// TIA Portal V19 export
VAR_GLOBAL   // PLC tag table "Tag table from XML_1"
   "At 1" AT %I0.0 : Bool;
   "At 2" AT %I0.1 : Bool;
   "At 3" AT %I0.2 : Bool;
   "At elevator" AT %I0.3 : Bool;
   "At entry" AT %I0.4 : Bool;
   "At exit" AT %I0.5 : Bool;
   "At 0 (low)" AT %I0.6 : Bool;
   "At 0 (high)" AT %I0.7 : Bool;
   "At 1 (low)" AT %I1.0 : Bool;
   "At 1 (high)" AT %I1.1 : Bool;
   "At 2 (low)" AT %I1.2 : Bool;
   "At 2 (high)" AT %I1.3 : Bool;
   "At 3 (low)" AT %I1.4 : Bool;
   "At 3 (high)" AT %I1.5 : Bool;
   Start AT %I1.6 : Bool;
   Reset AT %I1.7 : Bool;
   Stop AT %I2.0 : Bool;
   "Emergency stop" AT %I2.1 : Bool;
   Auto AT %I2.2 : Bool;
   "Diffuse Sensor 0" AT %I2.3 : Bool;
   "Diffuse Sensor 1" AT %I2.4 : Bool;
   "Diffuse Sensor 2" AT %I2.5 : Bool;
   "Diffuse Sensor 3" AT %I2.6 : Bool;
   "Conveyor 0" AT %Q0.0 : Bool;
   "Conveyor 1" AT %Q0.1 : Bool;
   "Conveyor 2" AT %Q0.2 : Bool;
   "Conveyor 3" AT %Q0.3 : Bool;
   "Exit conveyor" AT %Q0.4 : Bool;
   Load AT %Q0.5 : Bool;
   Unload AT %Q0.6 : Bool;
   Up AT %Q0.7 : Bool;
   Down AT %Q1.0 : Bool;
   Slow AT %Q1.1 : Bool;
   "Warning light" AT %Q1.2 : Bool;
   "Start light" AT %Q1.3 : Bool;
   "Reset light" AT %Q1.4 : Bool;
   "Stop light" AT %Q1.5 : Bool;
   "Floor 1" AT %Q1.6 : Bool;
   "Floor 2" AT %Q1.7 : Bool;
   "Floor 3" AT %Q2.0 : Bool;
   "Green 1" AT %Q2.1 : Bool;
   "Yellow 1" AT %Q2.2 : Bool;
   "Red 1" AT %Q2.3 : Bool;
   "Green 2" AT %Q2.4 : Bool;
   "Yellow 2" AT %Q2.5 : Bool;
   "Red 2" AT %Q2.6 : Bool;
   "Green 3" AT %Q2.7 : Bool;
   "Yellow 3" AT %Q3.0 : Bool;
   "Red 3" AT %Q3.1 : Bool;
   Display AT %QD100 : DInt;
END_VAR
